INTERFACE I_Event EXTENDS I_Object

METHOD PUBLIC M_Abort : BOOL
VAR_INPUT
	Message:				STRING(255);
	ID:						ID;
END_VAR
END_METHOD

METHOD PUBLIC M_AddBOOL
VAR_INPUT
	Value: 	BOOL;
END_VAR
END_METHOD

METHOD PUBLIC M_AddINT
VAR_INPUT
	Value: 	LINT;
END_VAR
END_METHOD

METHOD PUBLIC M_AddREAL
VAR_INPUT
	Value: 	Lreal;
	Decimals: INT;
END_VAR
END_METHOD

METHOD PUBLIC M_AddSTRING
VAR_INPUT
	Value: STRING(255);
END_VAR
END_METHOD

METHOD PUBLIC M_Debug : BOOL
VAR_INPUT
	Message:				STRING(255);
END_VAR
END_METHOD

METHOD PUBLIC M_Information : BOOL
VAR_INPUT
	Message:				STRING(255);
	ID:						ID;
END_VAR
END_METHOD

METHOD PUBLIC M_Stop : BOOL
VAR_INPUT
	Message:				STRING(255);
	ID:						ID;
END_VAR
END_METHOD

METHOD PUBLIC M_StopCycle : BOOL
VAR_INPUT
	Message:				STRING(255);
	ID:						ID;
END_VAR
END_METHOD

METHOD PUBLIC M_Warning : BOOL
VAR_INPUT
	Message:				STRING(255);
	ID:						ID;
END_VAR
END_METHOD

PROPERTY PUBLIC P_Logger : I_Logger
GET
END_GET
SET
END_SET
END_PROPERTY

END_INTERFACE

(* stored: Version 1.1.0.1
   Itf I_Event: Id {86200139-fcb7-4d9e-9f1b-6b3e88f31cc6}
   Method M_Abort: Id {7ce1cd66-528d-482d-8b65-9ae3dbff679e}
   Method M_AddBOOL: Id {6fc486ba-f21e-0356-3f27-fe3c53264131}
   Method M_AddINT: Id {a79ade02-7143-0a56-3ea5-b2c5275bc535}
   Method M_AddREAL: Id {ebc5d459-c769-0e97-2a4f-b9373812d338}
   Method M_AddSTRING: Id {3ed3c97e-76ae-02a4-026a-a11cdc8c444d}
   Method M_Debug: Id {de8efd53-16f5-0334-02e3-fdd0e4bf084c}
   Method M_Information: Id {a0df6aac-21ac-0b65-3426-2421a14ee702}
   Method M_Stop: Id {afad8492-19cf-0779-1a83-3ea67e573ec9}
   Method M_StopCycle: Id {941c4bf1-5b90-0130-09bd-59407d728f49}
   Method M_Warning: Id {ae861465-4d88-0ffb-03b6-6d69b34da892}
   Property P_Logger: Id {79c5886e-8d4f-463a-a8f3-e7a7286bafb7}
   Get Get: Id {d72a2fbe-a299-4aee-94b4-9d545177e15c}
   Set Set: Id {769c2202-eaa4-4a8d-ad42-86a0c8601e68} *)
